FUNCTION_BLOCK NeredaReactor (* CAT Function Block Type *)
  (* Standard: 61499-2 *)
  (* Version 0.0, 6/7/2026, Schneider Electric, template *)
  PACKAGE SE.Nereda;
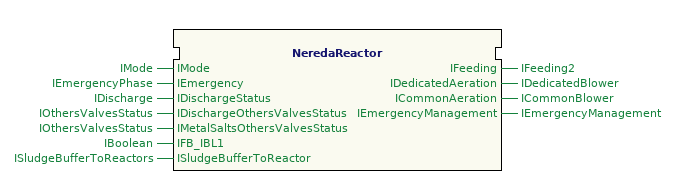
  SOCKETS
    IMode : IMode;
    IEmergency : IEmergencyPhase;
    IDischargeStatus : IDischarge; (* Phase Sludge Discharge Status *)
    IDischargeOthersValvesStatus : IOthersValvesStatus; (* Phase Sludge Discharge Status *)
    IMetalSaltsOthersValvesStatus : IOthersValvesStatus;
    IFB_IBL1 : IBoolean;
    ISludgeBufferToReactor : ISludgeBufferToReactors;
  END_SOCKETS
  PLUGS
    IFeeding : IFeeding2; (* Phase Feed Cmd *)
    IDedicatedAeration : IDedicatedBlower; (* Phase Aerate Cmd *)
    ICommonAeration : ICommonBlower;
    IEmergencyManagement : IEmergencyManagement;
  END_PLUGS
  (* 01 - FUNCTIONNAL INPUT INTERFACE *)
  (* 00 - INITIALIZATION *)
  (* 05 - LOGIC *)
  (* 06 - HMI INTERFACE *)
  (* 03 - FIELD INTERFACE *)
  (* 02 - FUNCTIONNAL OUTPUT INTERFACE *)
  (* Reactor Logic *)
  (* 04 - CHILDREN *)
  (* 4A - TYPICALS *)
  (* 07- REACTOR ALARM *)
  (* Actuators Tags : - Feed valve :                                  AV4x101 - Lower level valve :                        AV4x102 - Air fill valve sludge discharge :    AV4x171 - Chemicals valve :                         AV4x108 - Discharge valve :                         AV4x103 - Vent aeration grid valve :             AV4x107 - Vent sludge grid valve :               AV4x172 *)
  FBS
    ReactorLogic : ReactorLogic;
    INIT : plcStart(Prio := 55, Delay := T#0ms);
    IThis : NeredaReactor_HMI(QI := TRUE);
    Actuators : ReactorActuators;
    Sensors : ReactorSensors;
    FeedAborted : ALARM_BIT(ACKTYPE_1 := 2, ACTIVE := TRUE, TYPE := 1);
    Insufficient_Sludge_Discharge : ALARM_BIT(ACKTYPE_1 := 2, TYPE := 1, ACTIVE := TRUE);
    AerateAborted : ALARM_BIT(ACKTYPE_1 := 2, ACTIVE := TRUE, TYPE := 1);
    SludgeDischargeAborted : ALARM_BIT(ACKTYPE_1 := 2, ACTIVE := TRUE, TYPE := 1);
    VentAborted : ALARM_BIT(ACKTYPE_1 := 2, ACTIVE := TRUE, TYPE := 1);
    Status : ReactorInStatus;
    LowerLevelAborted : ALARM_BIT(ACKTYPE_1 := 2, TYPE := 1, ACTIVE := TRUE);
    MetalDosingAborted : ALARM_BIT(ACKTYPE_1 := 2, ACTIVE := TRUE, TYPE := 1);
    VentAerationGridAborted : ALARM_BIT(ACKTYPE_1 := 2, ACTIVE := TRUE, TYPE := 1);
    VentSludgeGridAborted : ALARM_BIT(ACKTYPE_1 := 2, ACTIVE := TRUE, TYPE := 1);
    DischargeOthersValvesStatus : MultiIOthersVlvStatus;
    DischargeStatus : MultiIDischarge;
  END_FBS
  EVENT_CONNECTIONS
    VentAborted.INITO TO Insufficient_Sludge_Discharge.INIT;
    INIT.FIRST_INIT TO IThis.76B3F71A0DA16C2E;
    INIT.REDO_INIT TO IThis.76B3F71A0DA16C2E;
    VentSludgeGridAborted.INITO TO INIT.ACK_FIRST;
    FeedAborted.CNF_INITDATA TO FeedAborted.REQ;
    VentSludgeGridAborted.INITO TO FeedAborted.REQ_INITDATA;
    VentSludgeGridAborted.INITO TO Insufficient_Sludge_Discharge.REQ_INITDATA;
    Insufficient_Sludge_Discharge.CNF_INITDATA TO Insufficient_Sludge_Discharge.REQ;
    FeedAborted.CNF_INITDATA TO FeedAborted.ACTIVATE;
    Insufficient_Sludge_Discharge.CNF_INITDATA TO Insufficient_Sludge_Discharge.ACTIVATE;
    IThis.740214A6EA51024E TO ReactorLogic.71EAA67E364772D7;
    Sensors.F5C2D5BE736233BA TO IThis.7DD2DECF8FCC304A;
    Sensors.D2EB091A02E78227 TO IThis.B3A782D12CC10E94;
    Sensors.C9AFBEBFCC954DBE TO ReactorLogic.73E8959D6DD12DB8;
    Sensors.C9AFBEBFCC954DBE TO ReactorLogic.EE40869F20F41A0D;
    ReactorLogic.9C75EF2A7C457F62 TO Sensors.INIT;
    ReactorLogic.CC035B2BAC15FA13 TO FeedAborted.REQ;
    ReactorLogic.D454B421DAC7C402 TO Insufficient_Sludge_Discharge.REQ;
    Sensors.INITO TO Actuators.INIT;
    Actuators.INITO TO FeedAborted.INIT;
    FeedAborted.INITO TO AerateAborted.INIT;
    AerateAborted.INITO TO SludgeDischargeAborted.INIT;
    SludgeDischargeAborted.INITO TO VentAborted.INIT;
    VentSludgeGridAborted.INITO TO AerateAborted.REQ_INITDATA;
    VentSludgeGridAborted.INITO TO SludgeDischargeAborted.REQ_INITDATA;
    VentSludgeGridAborted.INITO TO VentAborted.REQ_INITDATA;
    AerateAborted.CNF_INITDATA TO AerateAborted.ACTIVATE;
    AerateAborted.CNF_INITDATA TO AerateAborted.REQ;
    SludgeDischargeAborted.CNF_INITDATA TO SludgeDischargeAborted.ACTIVATE;
    SludgeDischargeAborted.CNF_INITDATA TO SludgeDischargeAborted.REQ;
    VentAborted.CNF_INITDATA TO VentAborted.ACTIVATE;
    VentAborted.CNF_INITDATA TO VentAborted.REQ;
    ReactorLogic.CC035B2BAC15FA13 TO AerateAborted.REQ;
    ReactorLogic.CC035B2BAC15FA13 TO SludgeDischargeAborted.REQ;
    ReactorLogic.CC035B2BAC15FA13 TO VentAborted.REQ;
    Status.4B81AC7A92DEAB20 TO IThis.2E53AF159919773C;
    ReactorLogic.CC035B2BAC15FA13 TO IThis.27392C087939011D;
    IThis.09BA6F3B382CD82A TO Status.42F2E1FCFC7E5858;
    ReactorLogic.A05CC99A535B95B5 TO Status.42F2E1FCFC7E5858;
    ReactorLogic.CC035B2BAC15FA13 TO Status.42F2E1FCFC7E5858;
    VentSludgeGridAborted.INITO TO LowerLevelAborted.REQ_INITDATA;
    LowerLevelAborted.CNF_INITDATA TO LowerLevelAborted.REQ;
    LowerLevelAborted.CNF_INITDATA TO LowerLevelAborted.ACTIVATE;
    Insufficient_Sludge_Discharge.INITO TO LowerLevelAborted.INIT;
    MetalDosingAborted.INITO TO VentAerationGridAborted.INIT;
    VentAerationGridAborted.INITO TO VentSludgeGridAborted.INIT;
    MetalDosingAborted.CNF_INITDATA TO MetalDosingAborted.REQ;
    MetalDosingAborted.CNF_INITDATA TO MetalDosingAborted.ACTIVATE;
    VentAerationGridAborted.CNF_INITDATA TO VentAerationGridAborted.ACTIVATE;
    VentAerationGridAborted.CNF_INITDATA TO VentAerationGridAborted.REQ;
    VentSludgeGridAborted.CNF_INITDATA TO VentSludgeGridAborted.ACTIVATE;
    VentSludgeGridAborted.CNF_INITDATA TO VentSludgeGridAborted.REQ;
    LowerLevelAborted.INITO TO MetalDosingAborted.INIT;
    VentSludgeGridAborted.INITO TO VentSludgeGridAborted.REQ_INITDATA;
    VentSludgeGridAborted.INITO TO VentAerationGridAborted.REQ_INITDATA;
    VentSludgeGridAborted.INITO TO MetalDosingAborted.REQ_INITDATA;
    ReactorLogic.CC035B2BAC15FA13 TO LowerLevelAborted.REQ;
    ReactorLogic.CC035B2BAC15FA13 TO MetalDosingAborted.REQ;
    ReactorLogic.CC035B2BAC15FA13 TO VentAerationGridAborted.REQ;
    ReactorLogic.CC035B2BAC15FA13 TO VentSludgeGridAborted.REQ;
  END_CONNECTIONS
  DATA_CONNECTIONS
    ReactorLogic.723242377777ED18 TO IThis.D3B631F986AC12CC;
    ReactorLogic.A103C4E7D0A13DD1 TO IThis.D85607DF26531674;
    ReactorLogic.40133CDA87CE6A95 TO IThis.5CCA6B03BE7B59C3;
    ReactorLogic.B8C8830DC2E6BD30 TO IThis.7A7006C2D6AE1D94;
    ReactorLogic.A0A7C43C0A43604D TO IThis.980CC725486FCDED;
    ReactorLogic.6AC7DFE8594172F8 TO IThis.34B07A5611C3DF95;
    Sensors.C4C37255D17EB4E6 TO IThis.2C8CF876EB93FE1F;
    Sensors.837F9EBED5615CB7 TO IThis.BCF24FABAD3885E7;
    Sensors.11E879B934FF1E2F TO IThis.E9D7938BD30E0CC0;
    Sensors.8D0251A007B7850C TO ReactorLogic.C020BB0D967C0574;
    Sensors.1CD741245A523D5B TO ReactorLogic.0832E74510330863;
    ReactorLogic.6620E61C8E6CE8CC TO Insufficient_Sludge_Discharge.INP;
    ReactorLogic.99BD1E64FA3D5F60 TO FeedAborted.INP;
    ReactorLogic.78DB1EA880F44385 TO AerateAborted.INP;
    ReactorLogic.6818BF610234DD80 TO SludgeDischargeAborted.INP;
    ReactorLogic.E993570727C49E8D TO VentAborted.INP;
    Status.5305838B7B9BBDAE TO IThis.765AD9E545DEE9A7;
    IThis.5C7F43170446F540 TO Status.1EBB7FA17C3153B3;
    ReactorLogic.205CB2F0624E2076 TO Status.C46408A3ABA13E13;
    ReactorLogic.87DB376EA1586B2F TO Status.27BB5B485A1EEF97;
    ReactorLogic.6B2A1EDEF7488E82 TO Status.50D65ED1800D8F1C;
    ReactorLogic.EEB23E7DBBAB1466 TO LowerLevelAborted.INP;
    ReactorLogic.F93B932F5CBBEB5B TO MetalDosingAborted.INP;
    ReactorLogic.71E4D5F5C0104FD8 TO VentAerationGridAborted.INP;
    ReactorLogic.6BDB004B1987AAA0 TO VentSludgeGridAborted.INP;
  END_CONNECTIONS
  ADAPTER_CONNECTIONS
    DischargeStatus.A052FE1D915AF2A9 TO ReactorLogic.0A33063DE6BF3285;
    DischargeOthersValvesStatus.A21F46DB29F1DA55 TO ReactorLogic.5FB5CD25010D5A2C;
    IMode TO ReactorLogic.98EF867CC88B438C;
    IEmergency TO ReactorLogic.01B158DA2C49BDF9;
    ReactorLogic.35768F64143690ED TO IFeeding;
    ReactorLogic.5FA056CAEE241C9B TO IDedicatedAeration;
    ReactorLogic.37E9E449EE210AC0 TO IEmergencyManagement;
    ReactorLogic.5508F8D8B77C7BD6 TO Actuators.CD98332339C83299;
    ReactorLogic.0572C576803DB81C TO Actuators.846EE90A7900F10A;
    Actuators.EAFAABEE532B9015 TO ReactorLogic.B7203F9117AD4DDE;
    Actuators.E75B3ACBCAEFEF2D TO ReactorLogic.A37105B35D314134;
    Actuators.CF266C966D280EC0 TO ReactorLogic.E14E3CF58A001DD1;
    Sensors.D12EBE3082937A2E TO ReactorLogic.F07B4F45A4C55A69;
    Sensors.D5D7A094F3CE5EF7 TO ReactorLogic.33C9571C798FF99B;
    Sensors.6BB9795C0E236086 TO ReactorLogic.F03AFC3BDFCB2B2A;
    ReactorLogic.64AF0FB1D2586385 TO ICommonAeration;
    ReactorLogic.1E74C4B8EB1EF069 TO Actuators.CC6CDF50573B1AD3;
    ReactorLogic.EF886F1C6170A76F TO Actuators.F0E19AA39D44C4EC;
    Actuators.F22AC61CBAB23CC3 TO ReactorLogic.F451F2337918C648;
    Actuators.0225F420D53D6628 TO ReactorLogic.6CB79B2DA3EDA778;
    Actuators.410905100E6B981B TO ReactorLogic.B62D1E88B1231AAE;
    Actuators.E7A2D69BF8C95A9F TO ReactorLogic.5F5D5D56D9BD8257;
    Actuators.B8F288117DB0B52C TO ReactorLogic.B679194CDF837D13;
    Actuators.CD9AA778407C3C3D TO ReactorLogic.93DF92981FD2F83C;
    Actuators.9117A8570E79370F TO ReactorLogic.CA5F07961CDBC5D6;
    Actuators.D53997F646C99AD5 TO ReactorLogic.5FA1BFCB059DB46C;
    Actuators.953934AD65EF1080 TO ReactorLogic.FE14E21ED8E970F7;
    Actuators.0C4BF007BE302AB2 TO ReactorLogic.D1EE3E20F5B96B90;
    IMetalSaltsOthersValvesStatus TO ReactorLogic.690D56B19FF35284;
    Actuators.97E797D2D271D3AF TO ReactorLogic.609074AB510D3EFE;
    Actuators.3B52B3F94C04F6EA TO ReactorLogic.E53F4A724AFC3278;
    ReactorLogic.F191ABE85B59B4E2 TO Actuators.B093A6B72B6914BA;
    Actuators.9CF3E36D56CE9FC3 TO ReactorLogic.219EBF9F30430550;
    IDischargeOthersValvesStatus TO DischargeOthersValvesStatus.AED0D7B5B9815986;
    IDischargeStatus TO DischargeStatus.30FC89504ED97C71;
    Actuators.53906814FAAC22DF TO ReactorLogic.1AF87AD2F89B108F;
    ReactorLogic.324A5000DAA4415A TO Actuators.46DEEED8E7202E26;
    IFB_IBL1 TO ReactorLogic.2967E886E2127911;
    ReactorLogic.6894E9469B776A22 TO Actuators.4A14CAC35978B412;
    ISludgeBufferToReactor TO ReactorLogic.F5015D649EBC5E65;
    Sensors.43985F38881B0D5C TO ReactorLogic.553E5C25E9E47E53;
    Actuators.34A354E22353BA57 TO ReactorLogic.A860951D83FEC1FB;
  END_CONNECTIONS
END_FUNCTION_BLOCK
